FUNCTION_BLOCK StopProgramTask EXTENDS TcoMitsubishiRoboticsTask
VAR

	_stopType: TcoAbstractions.eTcoRoboticsStopType;
END_VAR



IF Execute() THEN
	IF _progress = 0 THEN
		IF NOT __ISVALIDREF(inoControl) THEN
			_varInfo :=__VARINFO(inoControl);
			Messenger.Programming(_sb.Clear().Append('<#Invalid reference: #>').Append(_varInfo.Symbol).ToString()).Pin();
		ELSIF NOT __ISVALIDREF(inoConfig) THEN                                                  
			_varInfo :=__VARINFO(inoConfig);                                                    
			Messenger.Programming(_sb.Clear().Append('<#Invalid reference: #>').Append(_varInfo.Symbol).ToString()).Pin();
		ELSIF NOT __ISVALIDREF(inoStatus) THEN                                                  
			_varInfo :=__VARINFO(inoStatus);                                                    
			Messenger.Programming(_sb.Clear().Append('<#Invalid reference: #>').Append(_varInfo.Symbol).ToString()).Pin();
			ELSE
			_progress := _progress + 1;
		END_IF

	END_IF
	
	IF _progress = 1 THEN
		inoControl.OpoerationEnable:=TRUE;
		_varInfo :=__VARINFO( inoStatus.State.OperationEnable);                                                
		THIS^.Messenger.OnCondition(_infoTimer.Q AND NOT inoStatus.State.OperationEnable).Warning(_sb.Clear().Append('<#Waiting for Operation enable signal! #>').Append(_varInfo.Symbol).ToString());
		IF  inoStatus.State.OperationEnable THEN
			_progress := _progress + 1;
		END_IF;
	END_IF;
	
	IF _progress = 2 THEN
	
		inoControl.AutoEnable:=TRUE;
		_varInfo :=__VARINFO( inoStatus.State.AutoEnable);                                                
		THIS^.Messenger.OnCondition(_infoTimer.Q AND NOT inoStatus.State.AutoEnable).Warning(_sb.Clear().Append('<#Waiting for Auto signal! #>').Append(_varInfo.Symbol).ToString());
		IF  inoStatus.State.AutoEnable THEN
			_progress := _progress + 1;
		END_IF;
	END_IF;
	
	IF _progress = 3 THEN
		inoControl.Stop:=TRUE ;
		inoControl.Start:=FALSE ;
		
		
		IF  inoStatus.State.Stop  THEN
				inoControl.Stop:=FALSE;
		END_IF
	END_IF;		
	
	
	_varInfo :=__VARINFO( inoStatus.State.Stop);                                                
	THIS^.Messenger.OnCondition(_infoTimer.Q AND NOT inoStatus.State.Stop)
		.Warning(_sb.Clear().Append('<# Waiting for signal: #>').Append(_varInfo.Symbol).Append('<# is OFF #>').ToString());
	
    DoneWhen( inoStatus.State.Stop );
    CallTimers(TRUE);
	
	THIS^.ThrowWhen(_errorTimer.Q);
END_IF

IF  THIS^.Error AND NOT _errorMessage.Pinned THEN
	THIS^.Restore();
END_IF

METHOD PUBLIC FB_init : BOOL
VAR_INPUT
    bInitRetains : BOOL; // if TRUE, the retain variables are initialized (warm start / cold start)
    bInCopyCode : BOOL; // if TRUE, the instance afterwards gets moved into the copy code (online change)
  	ParentObject : ITcoObject;	
END_VAR
END_METHOD

METHOD INTERNAL InvokeWithParams : ITcoTaskStatus
VAR_INPUT
	inStopType : eTcoRoboticsStopType;
END_VAR
_stopType := inStopType;
InvokeWithParams := THIS^.Invoke();
END_METHOD

(*~
	<docu>
		<summary>
			Executes when task is aborted.
		</summary>			
	</docu>	
~*)
METHOD PROTECTED OnAbort
IF  __ISVALIDREF(inoStatus) THEN   THIS^.inoStatus.ActionDescription := '<#Stop program was aborted, while not yet completed!#>';END_IF; 
inoControl.Stop:=FALSE;
END_METHOD

(*~
	<docu>
		<summary>
			Executes when task reaches the ```Done``` state .
		</summary>			
	</docu>	
~*)
METHOD PROTECTED OnDone
IF  __ISVALIDREF(inoStatus) THEN  THIS^.inoStatus.ActionDescription := '<#Stop program was completed successfully.#>';END_IF; 
_progress:=0;
END_METHOD

(*~
	<docu>
		<summary>
			Executes when task reaches the ```Error``` state.
>
		</summary>			
	</docu>	
~*)
METHOD PROTECTED OnError
VAR
	description: STRING;
END_VAR
THIS^.inoStatus.ActionDescription := '<#Stopping program with error.#>';
IF  __ISVALIDREF(inoStatus) THEN   THIS^.inoStatus.ActionDescription := description; END_IF;
THIS^._errorMessage.Error(_sb.Clear().Append(description).Append(' To restore acknowledge this alarm.').ToString()).Pin();
END_METHOD

METHOD PROTECTED OnStart
IF  __ISVALIDREF(inoStatus) THEN  THIS^.inoStatus.ActionDescription := '<#Stopping program started.#>'; END_IF; 
CallTimers(FALSE);
END_METHOD

(*~
	<docu>
		<summary>
			Restores this instance to the Ready state. Can be called explicitly or from within one of the restore mechanisms.
			<para>
				See also <see cref="PlcDocu.TcoCore.TcoTask.AutoRestorable()"/>
			</para>
		</summary>			
	</docu>	
~*)
METHOD Restore : ITcoRestorable
SUPER^.Restore();
inoControl.Stop:=FALSE;
END_METHOD

END_FUNCTION_BLOCK

(* stored: Version 1.1.0.1, ProductVersion 3.1.4024.12
   POU StopProgramTask: Id {7f6fa0f4-1e67-09be-1510-ab5b9cbeafa8}, SpecialFunc None
   Method FB_init: Id {3d8584f4-0200-0901-0ce9-483e90f1bbb5}
   Method InvokeWithParams: Id {d4e019c9-2c9b-040e-1c25-8abe6ed06768}
   Method OnAbort: Id {046f8aff-1212-06a5-1d13-bebc774fba42}
   Method OnDone: Id {de5075e0-1242-019a-168a-c1a76ccb7474}
   Method OnError: Id {73684542-e5c2-0145-39a5-1b6075d0c64f}
   Method OnStart: Id {4d5f5f9c-f516-010a-06db-ff3360ae586f}
   Method Restore: Id {0e42bf55-c64b-0c02-3714-261828d547ec} *)
